//{attribute 'pack_mode' := '8'}
TYPE ST_PCMProduct :
STRUCT
	EndMarket			: 	STRING(10);
	BatchID			:	T_CodeBATCH;
	ProductionOrder	:	T_CodePO;
	OuterType			: 	STRING(5);
	PITCode			:	T_CodePIT;

	HierarchyDataList	:	ST_HierarchyDataList;

	UoM				:	STRING(5);
END_STRUCT
END_TYPE

(* stored: Version 1.1.0.1
   DUT ST_PCMProduct: Id {aa06421f-be09-4d70-963e-ed1d9371da0a} *)
